PROGRAM MAIN
VAR
	//Test : St_Event ;
	buton : BOOL := FALSE ;
	
	eEventType1 : E_EventType := E_EventType.Alarm ;
	eEventSeverity1 : TcEventSeverity := TcEventSeverity.Error ;
	nEventIdentiy1 : UDINT := 42 ;
	sEventText1 : STRING (255) := 'This is a scary event' ;
	
	CsvPersistentEventStorage : FB_CsvPersistentEventStorage ;
	EventLogger : FB_EventLogger(CsvPersistentEventStorage) ;
	
	
END_VAR


IF buton THEN
	EventLogger.AddEvent(eEventType1, eEventSeverity1, nEventIdentiy1, sEventText1);
	buton := FALSE ;
 
END_IF

CsvPersistentEventStorage();

END_PROGRAM

(* stored: Version 1.1.0.1, ProductVersion 3.1.4024.12
   POU MAIN: Id {34582b17-7265-45bc-a906-db94733f1e07}, SpecialFunc None *)
